VAR_GLOBAL CONSTANT
  MAX_PROCESS       : UINT := 13;
END_VAR
{attribute 'qualified_only'}
VAR_GLOBAL
  Simulation        : ARRAY[1..MAX_PROCESS] OF fb_Simulation;
END_VAR

(* stored: Version 1.1.0.1
   GVL GVL_APPLICATION: Id {ef5c8ee7-19c1-4689-9600-6bba8e125d3a} *)
